TYPE ST_INPUT_IO :
STRUCT
	io AT%I*:ARRAY [1..16] OF BOOL;
END_STRUCT
END_TYPE

(* stored: Version 1.1.0.1, ProductVersion 3.1.4024.4
   DUT ST_INPUT_IO: Id {952db6f6-f88b-4ece-b9ca-59bfd9ef9652} *)
